(* PLC project TEST.project, CODESYS CODESYS V3.5 SP3 Patch 7 *)
(* stored: creationDateTime 2013-12-18T19:56:41.0388077, modificationDateTime 2013-12-18T19:56:09.7450178 *)

FUNCTION_BLOCK Endlagenschalter
  VAR
    bet : INT;
    tigt : INT;
    unbet : INT;
    Signal : INT;
    Drehung : INT;
  END_VAR

INITIAL_STEP Endlagenschalter bereit:
END_STEP
TRANSITION FROM Endlagenschalter bereit TO Motor Signal AUS
  := betätigt;
END_TRANSITION
TRANSITION FROM Endlagenschalter bereit TO Motor Signal AN
  := unbetätigt;
END_TRANSITION
STEP Motor Signal AUS:
END_STEP
TRANSITION FROM Motor Signal AUS TO Init
  := Signal Drehung;
END_TRANSITION
STEP Motor Signal AN:
END_STEP
TRANSITION FROM Motor Signal AN TO Init
  := betätigt;
END_TRANSITION
END_FUNCTION_BLOCK
